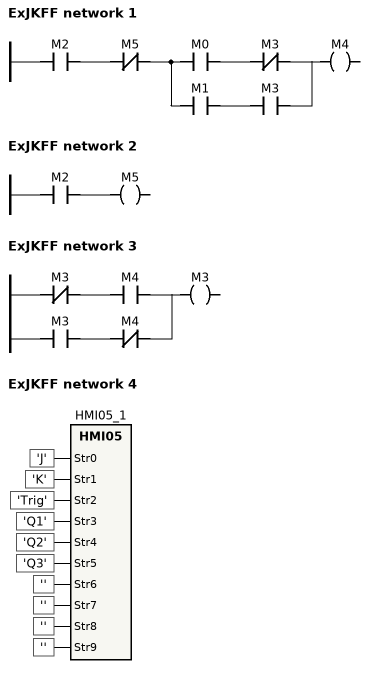
(* [picture p24: structured ladder/FBD of ExJKFF, networks 1 to 4] *)
(* network 1 *)
_p1 := M2 AND NOT M5;
M4 := (_p1 AND M0 AND NOT M3) OR (_p1 AND M1 AND M3);
(* network 2 *)
M5 := M2;
(* network 3 *)
M3 := (NOT M3 AND M4) OR (M3 AND NOT M4);
(* network 4 *)
HMI05_1(Str0 := 'J', Str1 := 'K', Str2 := 'Trig', Str3 := 'Q1', Str4 := 'Q2', Str5 := 'Q3', Str6 := '', Str7 := '', Str8 := '', Str9 := '');
END_PROGRAM

PROGRAM ExTFF
VAR
  HMI05_1 : HMI05;
END_VAR
(* structured ladder/FBD written out as ST: instructions are called as NAME(EN, inputs, outputs); _pN, _eN, _tN stand for wires *)
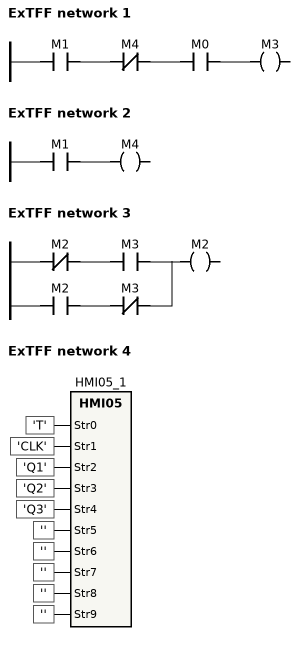
(* network 1 *)
M3 := M1 AND NOT M4 AND M0;
(* network 2 *)
M4 := M1;
(* network 3 *)
M2 := (NOT M2 AND M3) OR (M2 AND NOT M3);
(* network 4 *)
HMI05_1(Str0 := 'T', Str1 := 'CLK', Str2 := 'Q1', Str3 := 'Q2', Str4 := 'Q3', Str5 := '', Str6 := '', Str7 := '', Str8 := '', Str9 := '');
END_PROGRAM
